TYPE ST_RecCtrl ://过程纠偏
STRUCT
    Cmd        :ST_RecCmd;
    Io            :ST_RecIo;
    Status      :ST_RecStatus;
END_STRUCT
END_TYPE

(* stored: Version 1.1.0.1, ProductVersion 3.1.4024.9
   DUT ST_RecCtrl: Id {33208703-ac7d-4fa5-bf3d-314d186b201a} *)
